{attribute addProperty BoxType "EK1960-0000-0019"}
{attribute addProperty Id "FSoE_InputsFSoE_Inputs_FED5CD6512015FSoE_OutputsFSoE_Outputs_931DC9C512015"}
{attribute addProperty CRC "3707820063"}
{attribute addProperty SizeInBites "240"}
{attribute addProperty SizeInBytes "30"}
TYPE Module_1_FSoE_DD00D81F :
STRUCT
	{attribute addProperty Name "FSoE_Inputs"}
	FSoE_Inputs  : FSoE_Inputs_FED5CD65;
	{attribute addProperty Name "FSoE_Outputs"}
	FSoE_Outputs  : FSoE_Outputs_931DC9C5;
END_STRUCT
END_TYPE

(* stored: Version 1.2.0.0, ProductVersion 3.1.4024.9
   DUT Module_1_FSoE_DD00D81F: Id {b4b66d28-081d-4fe9-bcf9-d31ee93ec9f3} *)
